KUKA KRL program: Comprobar_camara.src, Comprobar_camara.dat

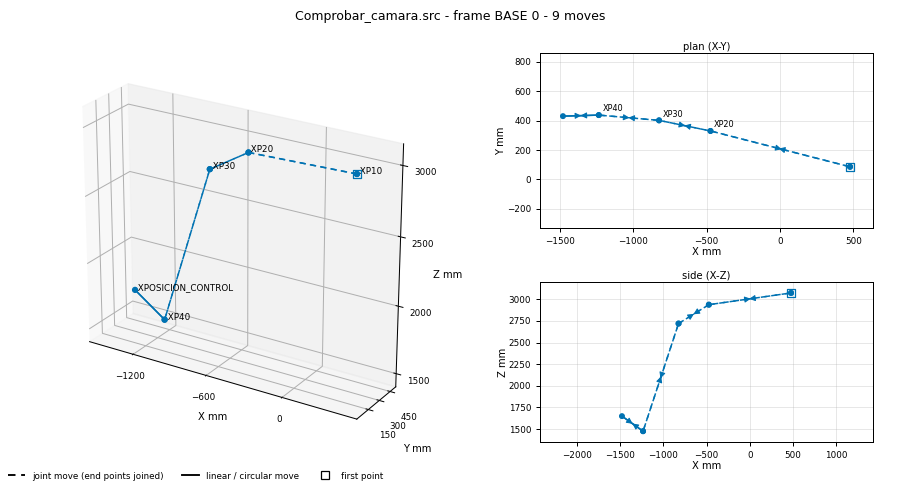
[picture p0: tool path of Comprobar_camara.src in frame BASE 0, 9 of 11 moves have a stored position in this frame; points joined in program order, loops and branches not executed]
--- Comprobar_camara.src ---
&ACCESS RVO1
&REL 42
&COMMENT PRG CONTROL CAMARA
&PARAM EDITMASK = *
&PARAM TEMPLATE = C:\KRC\Roboter\Template\vorgabe
&PARAM DISKPATH = KRC:\R1\Program\MAFELEC
DEF Comprobar_camara( )
;FOLD INI;%{PE}
  ;FOLD BASISTECH INI
    GLOBAL INTERRUPT DECL 3 WHEN $STOPMESS==TRUE DO IR_STOPM ( )
    INTERRUPT ON 3
    BAS (#INITMOV,0 )
  ;ENDFOLD (BASISTECH INI)
;FOLD SPOTTECH INI
USERSPOT(#INIT)
;ENDFOLD (SPOTTECH INI)
;FOLD GRIPPERTECH INI
USER_GRP(0,DUMMY,DUMMY,GDEFAULT)
;ENDFOLD (GRIPPERTECH INI)
  ;FOLD USER INI
    ;Make your modifications here

  ;ENDFOLD (USER INI)
;ENDFOLD (INI)
;################################################
; PROYECTO: MAFELEC PLANTA DE BATERIAS
; ROBOT: 121_R1
; PROGRAMA: CHEQUEO  DE CONTROL CAMARA
; CREADO POR: Alejandro Company(zaisor robotics)
; FECHA: 28-NOVIEMBRE-2022
; MODIFICADO POR:
; FECHA MODIFICACION: 17-ENERO-2023
;################################################

;FOLD PTP HOME  Vel= 100 % DEFAULT;%{PE}%MKUKATPBASIS,%CMOVE,%VPTP,%P 1:PTP, 2:HOME, 3:, 5:100, 7:DEFAULT
$BWDSTART = FALSE
PDAT_ACT=PDEFAULT
FDAT_ACT=FHOME
BAS (#PTP_PARAMS,100 )
$H_POS=XHOME
PTP  XHOME
;ENDFOLD

Empujador(1,"R",TRUE)
Empujador(2,"R",TRUE)
Pines("R")

;FOLD PTP P10 CONT Vel=20 % M Tool[9]:T_Gripper1_Vacio Base[0];%{PE}%R 8.3.48,%MKUKATPBASIS,%CMOVE,%VPTP,%P 1:PTP, 2:P10, 3:C_DIS, 5:20, 7:M
$BWDSTART=FALSE
PDAT_ACT=PM
FDAT_ACT=FP10
BAS(#PTP_PARAMS,20)
PTP XP10 C_DIS
;ENDFOLD
;FOLD PTP P20 CONT Vel=20 % M Tool[9]:T_Gripper1_Vacio Base[0];%{PE}%R 8.3.48,%MKUKATPBASIS,%CMOVE,%VPTP,%P 1:PTP, 2:P20, 3:C_DIS, 5:20, 7:M
$BWDSTART=FALSE
PDAT_ACT=PM
FDAT_ACT=FP20
BAS(#PTP_PARAMS,20)
PTP XP20 C_DIS
;ENDFOLD
;FOLD PTP P30 CONT Vel=20 % M Tool[9]:T_Gripper1_Vacio Base[0];%{PE}%R 8.3.48,%MKUKATPBASIS,%CMOVE,%VPTP,%P 1:PTP, 2:P30, 3:C_DIS, 5:20, 7:M
$BWDSTART=FALSE
PDAT_ACT=PM
FDAT_ACT=FP30
BAS(#PTP_PARAMS,20)
PTP XP30 C_DIS
;ENDFOLD
;FOLD PTP P40 CONT Vel=20 % M Tool[9]:T_Gripper1_Vacio Base[0];%{PE}%R 8.3.48,%MKUKATPBASIS,%CMOVE,%VPTP,%P 1:PTP, 2:P40, 3:C_DIS, 5:20, 7:M
$BWDSTART=FALSE
PDAT_ACT=PM
FDAT_ACT=FP40
BAS(#PTP_PARAMS,20)
PTP XP40 C_DIS
;ENDFOLD


;FOLD LIN POSICION_CONTROL Vel=0.1 m/s M Tool[9]:T_Gripper1_Vacio Base[0];%{PE}%R 8.3.48,%MKUKATPBASIS,%CMOVE,%VLIN,%P 1:LIN, 2:POSICION_CONTROL, 3:, 5:0.1, 7:M
$BWDSTART=FALSE
LDAT_ACT=LM
FDAT_ACT=FPOSICION_CONTROL
BAS(#CP_PARAMS,0.1)
LIN XPOSICION_CONTROL
;ENDFOLD
FOTITO()

O_SERVP=TRUE


;ESPERA PERMISO RETORNO A HOME
WAIT FOR I_RETHP
O_SERVP=FALSE

;FOLD LIN P40 Vel=0.5 m/s M Tool[9]:T_Gripper1_Vacio Base[0];%{PE}%R 8.3.48,%MKUKATPBASIS,%CMOVE,%VLIN,%P 1:LIN, 2:P40, 3:, 5:0.5, 7:M
$BWDSTART=FALSE
LDAT_ACT=LM
FDAT_ACT=FP40
BAS(#CP_PARAMS,0.5)
LIN XP40
;ENDFOLD


;FOLD PTP P30 CONT Vel=20 % M Tool[9]:T_Gripper1_Vacio Base[0];%{PE}%R 8.3.48,%MKUKATPBASIS,%CMOVE,%VPTP,%P 1:PTP, 2:P30, 3:C_DIS, 5:20, 7:M
$BWDSTART=FALSE
PDAT_ACT=PM
FDAT_ACT=FP30
BAS(#PTP_PARAMS,20)
PTP XP30 C_DIS
;ENDFOLD
;FOLD PTP P20 CONT Vel=20 % M Tool[9]:T_Gripper1_Vacio Base[0];%{PE}%R 8.3.48,%MKUKATPBASIS,%CMOVE,%VPTP,%P 1:PTP, 2:P20, 3:C_DIS, 5:20, 7:M
$BWDSTART=FALSE
PDAT_ACT=PM
FDAT_ACT=FP20
BAS(#PTP_PARAMS,20)
PTP XP20 C_DIS
;ENDFOLD
;FOLD PTP P10 CONT Vel=20 % M Tool[9]:T_Gripper1_Vacio Base[0];%{PE}%R 8.3.48,%MKUKATPBASIS,%CMOVE,%VPTP,%P 1:PTP, 2:P10, 3:C_DIS, 5:20, 7:M
$BWDSTART=FALSE
PDAT_ACT=PM
FDAT_ACT=FP10
BAS(#PTP_PARAMS,20)
PTP XP10 C_DIS
;ENDFOLD

;FOLD PTP HOME  Vel= 100 % DEFAULT;%{PE}%MKUKATPBASIS,%CMOVE,%VPTP,%P 1:PTP, 2:HOME, 3:, 5:100, 7:DEFAULT
$BWDSTART = FALSE
PDAT_ACT=PDEFAULT
FDAT_ACT=FHOME
BAS (#PTP_PARAMS,100 )
$H_POS=XHOME
PTP  XHOME
;ENDFOLD

END

DEF FOTITO()

; INICIALIZACION CAMARA
 INPICKER_Handler.DataToSend.command=0
 INPICKER_Handler.DataToSend.GraspConfirmation=0
 WAIT FOR (INPICKER_Handler.DataReceived.state==0)

; Camara siempre 2
 INPICKER_Handler.DataToSend.CameraID=0

; contendor igual al numero de bandeja
 INPICKER_Handler.DataToSend.ContainerID=12
 INPICKER_Handler.DataToSend.partid=0
 INPICKER_Handler.DataToSend.GraspConfirmation=0
 WAIT SEC 0.2

; DISPARO FOTO
 INPICKER_Handler.DataToSend.command=1

; ESPERA FOTO REALIZADA
 WAIT FOR (INPICKER_Handler.DataReceived.state==30) OR (INPICKER_Handler.DataReceived.state==-1)
wait sec 2
IF (INPICKER_handler.datareceived.state==-1 ) OR (INPICKER_Handler.DataReceived.ObjectsGraspable<=0) THEN

   ;*********************************
   ;FALLO FOTO -1, NO VE EL OBJETO
   WAIT FOR FALSE
   ;*********************************

ENDIF

IF (INPICKER_Handler.DataReceived.state==30) THEN

   IF FALSE THEN
      FRAME_MASTER=INPICKER_Handler.DataReceived.PartsToGrasp0.Position
   ENDIF

   FRAMEAUX=INPICKER_Handler.DataReceived.PartsToGrasp0.Position

   WAIT FOR ((ABS((FRAME_MASTER.X)-(FRAMEAUX.X)))<10) ;LIMITE EN X DENTRO DE RANGO
   WAIT FOR ((ABS((FRAME_MASTER.Y)-(FRAMEAUX.y)))<10) ;LIMITE EN Y DENTRO DE RANGO
   WAIT FOR ((ABS((FRAME_MASTER.Z)-(FRAMEAUX.z)))<10) ;LIMITE EN Z DENTRO DE RANGO
   WAIT FOR ((ABS((FRAME_MASTER.A)-(FRAMEAUX.a)))<10) ;LIMITE EN A DENTRO DE RANGO
   WAIT FOR ((ABS((FRAME_MASTER.B)-(FRAMEAUX.b)))<10) ;LIMITE EN B DENTRO DE RANGO
   WAIT FOR ((ABS((FRAME_MASTER.C)-(FRAMEAUX.c)))<10) ;LIMITE EN C DENTRO DE RANGO

ENDIF




END

--- Comprobar_camara.dat ---
&ACCESS RVO1
&REL 42
&COMMENT PRG CONTROL CAMARA
&PARAM EDITMASK = *
&PARAM TEMPLATE = C:\KRC\Roboter\Template\vorgabe
&PARAM DISKPATH = KRC:\R1\Program\MAFELEC
DEFDAT  Comprobar_camara
;FOLD EXTERNAL DECLARATIONS;%{PE}%MKUKATPBASIS,%CEXT,%VCOMMON,%P
;FOLD GRIPPERTECH EXT
EXT  H50 (INT  :IN,INT  :IN,INT  :IN,GRP_TYP  :IN )
;ENDFOLD (GRIPPERTECH EXT)
;FOLD SPOTTECH EXT
EXT  USERSPOT (S_COMMAND  :IN,SPOT_TYPE  :IN )
;ENDFOLD (SPOTTECH EXT)
;FOLD BASISTECH EXT;%{PE}%MKUKATPBASIS,%CEXT,%VEXT,%P
EXT  BAS (BAS_COMMAND  :IN,REAL  :IN )
DECL INT SUCCESS
;ENDFOLD (BASISTECH EXT)
;FOLD USER EXT;%{E}%MKUKATPUSER,%CEXT,%VEXT,%P
;Make your modifications here

;ENDFOLD (USER EXT)
;ENDFOLD (EXTERNAL DECLARATIONS)
DECL BASIS_SUGG_T LAST_BASIS={POINT1[] "P0                      ",POINT2[] "P0                      ",CP_PARAMS[] "CPDAT0                  ",PTP_PARAMS[] "PDAT0                   ",CONT[] "                        ",CP_VEL[] "2.0                     ",PTP_VEL[] " 100                    ",SYNC_PARAMS[] "SYNCDAT                 ",SPL_NAME[] "S0                      ",A_PARAMS[] "ADAT0                   "}
DECL E6POS XP1={X -1423.22278,Y 12.1733541,Z 595.070862,A 13.3003607,B 1.31921577,C -179.688721,S 2,T 11,E1 0.0,E2 0.0,E3 0.0,E4 0.0,E5 0.0,E6 0.0}
DECL FDAT FP1={TOOL_NO 9,BASE_NO 0,IPO_FRAME #BASE,POINT2[] " ",TQ_STATE FALSE}
DECL PDAT PPDAT1={VEL 100.000,ACC 100.000,APO_DIST 100.000,APO_MODE #CDIS,GEAR_JERK 50.0000,EXAX_IGN 0}
DECL E6POS XP10={X 477.041595,Y 86.2656479,Z 3074.07861,A -151.431854,B -26.5239220,C 5.04246378,S 7,T 27,E1 0.0,E2 0.0,E3 0.0,E4 0.0,E5 0.0,E6 0.0}
DECL FDAT FP10={TOOL_NO 9,BASE_NO 0,IPO_FRAME #BASE,POINT2[] " ",TQ_STATE FALSE}
DECL E6POS XP20={X -473.112488,Y 330.224060,Z 2938.42798,A -159.082184,B -30.9372654,C 55.3069801,S 6,T 27,E1 0.0,E2 0.0,E3 0.0,E4 0.0,E5 0.0,E6 0.0}
DECL FDAT FP20={TOOL_NO 9,BASE_NO 0,IPO_FRAME #BASE,POINT2[] " ",TQ_STATE FALSE}
DECL PDAT PM={VEL 100.000,ACC 50.0000,APO_DIST 100.000,APO_MODE #CDIS,GEAR_JERK 50.0000,EXAX_IGN 0}
DECL E6POS XP30={X -823.312805,Y 402.331848,Z 2720.40503,A -169.181305,B -23.5042057,C 82.1668549,S 6,T 27,E1 0.0,E2 0.0,E3 0.0,E4 0.0,E5 0.0,E6 0.0}
DECL FDAT FP30={TOOL_NO 9,BASE_NO 0,IPO_FRAME #BASE,POINT2[] " ",TQ_STATE FALSE}
DECL E6POS XP40={X -1233.62781,Y 438.195435,Z 1475.76819,A -167.316,B 34.6241,C 98.8769150,S 6,T 27,E1 0.0,E2 0.0,E3 0.0,E4 0.0,E5 0.0,E6 0.0}
DECL FDAT FP40={TOOL_NO 9,BASE_NO 0,IPO_FRAME #BASE,POINT2[] " ",TQ_STATE FALSE}
DECL E6POS XPOSICION_CONTROL={X -1477.56238,Y 431.007294,Z 1649.92090,A -178.076675,B 34.6241112,C 98.8769150,S 6,T 27,E1 0.0,E2 0.0,E3 0.0,E4 0.0,E5 0.0,E6 0.0}
DECL FDAT FPOSICION_CONTROL={TOOL_NO 9,BASE_NO 0,IPO_FRAME #BASE,POINT2[] " ",TQ_STATE FALSE}
DECL LDAT LM={VEL 2.00000,ACC 25.0000,APO_DIST 100.000,APO_FAC 50.0000,AXIS_VEL 100.000,AXIS_ACC 100.000,ORI_TYP #VAR,CIRC_TYP #BASE,JERK_FAC 50.0000,GEAR_JERK 50.0000,EXAX_IGN 0}
DECL E6POS XP41={X -1423.22278,Y 12.1733541,Z 595.070862,A 13.3003607,B 1.31921577,C -179.688721,S 2,T 11,E1 0.0,E2 0.0,E3 0.0,E4 0.0,E5 0.0,E6 0.0}
DECL FDAT FP41={TOOL_NO 9,BASE_NO 0,IPO_FRAME #BASE,POINT2[] " ",TQ_STATE FALSE}
DECL E6POS XP42={X -1423.22278,Y 12.1733541,Z 595.070862,A 13.3003607,B 1.31921577,C -179.688721,S 2,T 11,E1 0.0,E2 0.0,E3 0.0,E4 0.0,E5 0.0,E6 0.0}
DECL FDAT FP42={TOOL_NO 9,BASE_NO 0,IPO_FRAME #BASE,POINT2[] " ",TQ_STATE FALSE}
DECL E6POS XP43={X -1423.22278,Y 12.1733541,Z 595.070862,A 13.3003607,B 1.31921577,C -179.688721,S 2,T 11,E1 0.0,E2 0.0,E3 0.0,E4 0.0,E5 0.0,E6 0.0}
DECL FDAT FP43={TOOL_NO 9,BASE_NO 0,IPO_FRAME #BASE,POINT2[] " ",TQ_STATE FALSE}
ENDDAT
